FUNCTION_BLOCK FB_READ_WITHOUT_TIMER

VAR_IN_OUT
	device: DEVICE;
	bExecute : BOOL;
END_VAR

VAR_OUTPUT
	execRead : BOOL := FALSE;
END_VAR

VAR
	
	fbTime   : FB_LocalSystemTime := ( bEnable := TRUE, dwCycle := 1 );
	
	readInputRegister : FB_MBReadInputRegs;
	readHoldingRegister : FB_MBReadRegs;
	

	//TYPE_ARR: ARRAY[1..2] OF STRING; 
	done: BOOL;
	
	timeOut: TIME := T#2S;
	readError : INT := 0;
	idError : UDINT;
	
	k: UINT;
	z: INT;
	
	switch_first_bit: INT;
	Aux_Dword: DWORD;
	
	j: INT := 0;
	
	timer: TON;
	delay : TIME := T#200MS;
	
	index : INT := 0;
	subState: INT;
	
	ReadInputs: INT;
END_VAR

	
IF bExecute AND NOT execRead THEN
	execRead 			:= TRUE;
	index 				:= 1;
	subState 			:= 6;
	
	readError 			:= 0;
	idError 			:= 0;
	
	device.CheckComm 	:= 0;

	fbTime();
	device.readTimestamp := DT_TO_UDINT( SYSTEMTIME_TO_DT( fbTime.systemTime ) );
END_IF



IF execRead THEN
	
	CASE subState OF
		
		1: 
			IF device.readParameter[index].id <> 0 THEN 
				
				subState := 2;
				
				IF device.readParameter[index].ModbusFunction = 3 THEN	
				
					readHoldingRegister(
						sIPAddr:= device.ServerIP, 
						nTCPPort:= device.ServerNumPort, 
						nUnitID:= device.ServerReadUnitID, 
						nQuantity:= device.readParameter[index].ReadQty, 
						nMBAddr:= device.readParameter[index].ReadAddress, 
						cbLength:= SIZEOF(WORD) * device.readParameter[index].ReadQty, 
						pDestAddr:= ADR(device.readParameter[index].AuxArr), 
						bExecute:= TRUE , 
						tTimeout:= timeOut, 
						bBusy=> device.readParameter[index].bBusy, 
						bError=>,
						(*bBusy=> device.ReadBusy,
						bError => device.ReadError,*)
						nErrId=>, 
						cbRead=> 
					);	
					
						

				ELSIF device.readParameter[index].ModbusFunction = 4 THEN
					
					
					readInputRegister(
						sIPAddr:= device.ServerIP, 
						nTCPPort:= device.ServerNumPort, 
						nUnitID:= device.ServerReadUnitID, 
						nQuantity:= device.readParameter[index].ReadQty, 
						nMBAddr:= device.readParameter[index].ReadAddress, 
						cbLength:= SIZEOF(WORD) * device.readParameter[index].ReadQty, 
						pDestAddr:= ADR(device.readParameter[index].AuxArr), 
						bExecute:= TRUE ,  
						tTimeout:= timeOut, 
						bBusy=> device.readParameter[index].bBusy, 
						bError=>,
						(*bBusy=> device.ReadBusy,
						bError => device.ReadError,*)
						nErrId=>, 
						cbRead=> 
					);
				
					
					
				END_IF
			ELSE
				subState := 3;
			END_IF
			
		2: 
			
			IF device.readParameter[index].ModbusFunction = 3 THEN
				
				IF readHoldingRegister.bError THEN
 					IF readHoldingRegister.nErrId = 1861 THEN
						idError := idError +1 ;
					END_IF
					
					device.CheckComm := readHoldingRegister.nErrId;
					
					device.readParameter[index].bError := TRUE; 
					subState := 4;
				ELSIF NOT readHoldingRegister.bBusy THEN
					
					device.readParameter[index].bError := FALSE;
					subState := 4;
				END_IF
				
			
				readHoldingRegister(bExecute:= FALSE);
			
				
				
			ELSIF device.readParameter[index].ModbusFunction = 4 THEN
				
				IF readInputRegister.bError THEN
					
					IF readInputRegister.nErrId = 1861 THEN
						idError := idError +1 ;
					END_IF
					
					device.CheckComm := readInputRegister.nErrId;
					
					device.readParameter[index].bError := TRUE;
					subState := 4;
				
				ELSIF NOT readInputRegister.bBusy THEN
					device.readParameter[index].bError := FALSE;
					subState := 4;
				END_IF
   
				readInputRegister(bExecute:= FALSE);
				
			END_IF
						
			
		3: 
			// EXIT
			execRead := FALSE; 
			
		4: // INCREMENT
			timer(IN:= NOT timer.Q, PT:= delay, Q=> , ET=> );
			
			IF timer.Q THEN
				index := index + 1;
				subState := 6;
			END_IF
			
		6: 	// CHECK
			IF index > device.readParameterCounter THEN
				subState := 3;
			ELSE 
				subState := 1;
			END_IF
		
		ELSE
			// Azioni di default se nessun altro caso corrisponde
			//errore := TRUE;
			execRead := FALSE;
			
	END_CASE;
END_IF

END_FUNCTION_BLOCK

(* stored: Version 1.1.0.1, ProductVersion 3.1.4024.13
   POU FB_READ_WITHOUT_TIMER: Id {498c4226-6a23-4ae3-aa41-4a1cf5837885}, SpecialFunc None *)
